TYPE ST_LAB_OuterData :
STRUCT
	sOuterCode			: T_MaxString;
	nOutersStatus		: INT;
	nOuterRejectID		: UINT;
	
	aPacks				: ARRAY[1..10] OF ST_LAB_PackData;
END_STRUCT
END_TYPE

(* stored: Version 1.1.0.1
   DUT ST_LAB_OuterData: Id {f0cd4794-bc66-4d38-98af-c1f6060b21ba} *)
